# EPICS substitutions: wedler_kreidel/wedls.subs
file ./db/wedler.db {

  { ELMNT = wedl01, DEVICE = kiste1, CHAN = 0 }
  { ELMNT = wedl02, DEVICE = kiste1, CHAN = 1 }
  { ELMNT = wedl03, DEVICE = kiste1, CHAN = 2 }

}
